(* LS Electric XG5000 project: XMC_CrossCoupled *)
(* project to test Cross Coupled functionality *)
(* PLC LSPLC *)
(* module base 0 slot 0: Input/Output Module:XMC-DN24 (DC 24V Input 8Points/TR output 16Points) *)
(* module base 0 slot 1: Internal Analog Input/Output:XMF-AH04E (A/D voltage/current 2 channels, D/A voltage 2 channels) *)
(* task Periodic Task: Kind=2 *)
(* task Initialization Task: Kind=1 *)
(* task NC Program: Kind=6 *)

PROGRAM Cross_Coupled_ST (* task: Scan Program *)
(* structured text example of cross-coupled control *)
VAR
    Axis1 : UINT := 1; (* variable for axis 1 *)
    Axis2 : UINT := 2; (* axis 2 variable *)
    Connect_ECAT : BOOL; (* command to execute EtherCAT network connection *)
    Disconnect_ECAT : BOOL; (* disconnect the ethercat network *)
    Execute_CrossCoupleOff : BOOL; (* command to turn off cross-coupled control for axis 1 and axis 2 *)
    Execute_CrossCoupleOn : BOOL; (* command to turn on cross-coupling of axis 1 and axis 2 *)
    Execute_Move : BOOL; (* execute move for axis 1 and axis 2 *)
    Execute_MPloopOff : BOOL; (* command to turn off master loop control for axis 1 and 2 *)
    Execute_MPloopOn : BOOL; (* command to execute master control position loop on *)
    INST_Axis1PloopOff : LS_MASTERPLOOPCONTROLOFF; (* fb to turn off master ploop control for axis 1 *)
    INST_Axis1PloopOn : LS_MASTERPLOOPCONTROLON; (* fb for axis 1 master ploop on *)
    INST_Axis1Relative : MC_MOVERELATIVE; (* relative move for axis 1 *)
    INST_Axis2PloopOff : LS_MASTERPLOOPCONTROLOFF; (* fb to turn off master ploop control for axis 2 *)
    INST_Axis2PloopOn : LS_MASTERPLOOPCONTROLON; (* fb for axis 2 master ploop on *)
    INST_Axis2Relative : MC_MOVERELATIVE; (* fb for relative move of axis 2 *)
    INST_Connect : LS_CONNECT; (* ethercat connect FB *)
    INST_CoupleOff : LS_CROSSCOUPLEDCONTROLOFF; (* fb to disable cross-coupling *)
    INST_CoupleOn : LS_CROSSCOUPLEDCONTROLON; (* fb for turning on cross coupling *)
    INST_Disconnect : LS_DISCONNECT; (* fb to disconnect ethercat network *)
    INST_PowerAll : MC_POWERALL; (* fb to power on all axes *)
    Power_On_Axes : BOOL; (* command to power on all axes *)
END_VAR
(* AutomationDirect.com has provided this code for convenience. This sample code is provided "as-is" with no expressed or implied warranty. 
 If the end user includes any of the sample code (in whole or part), it is the user's responsibility to completely modify, integrate, and test any code to ensure it meets all system and 
 safety requirements for the intended application or system. *)

//Function block Calls
INST_Connect(Execute:=Connect_ECAT, ErrorID=>INST_Connect.ErrorID);
INST_Disconnect(Execute:=Disconnect_ECAT, ErrorID=>INST_Disconnect.ErrorID);

INST_PowerAll(Enable:=Power_On_Axes, Status=>INST_PowerAll.Status, Valid=>INST_PowerAll.Valid, ErrorID=>INST_PowerAll.ErrorID);

INST_Axis1PloopOn(Execute:=Execute_MPloopOn, Axis:=Axis1, P_Gain:=1100.0, I_Gain:=600.0, VelFF_Gain:=10000.0, CtrlLimit:=100000000.0, InControl=>INST_Axis1PloopOn.InControl, ErrorID=>INST_Axis1PloopOn.ErrorID);
INST_Axis2PloopOn(Execute:=Execute_MPloopOn, Axis:=Axis2, P_Gain:=1100.0, I_Gain:=600.0, VelFF_Gain:=10000.0, CtrlLimit:=100000000.0, InControl=>INST_Axis2PloopOn.InControl, ErrorID=>INST_Axis2PloopOn.ErrorID);

INST_CoupleOn(Execute:=Execute_CrossCoupleOn, Axis:=Axis1, PairAxis:=Axis2, P_Gain:=1100.0, SlaveMode:=FALSE, InControl=>INST_CoupleOn.InControl, ErrorID=>INST_CoupleOn.ErrorID);

INST_Axis1Relative(Execute:=Execute_Move, Axis:=Axis1, ContinuousUpdate:=FALSE, Distance:=50000.0, Velocity:=500000.0, 
	Acceleration:=500000.0, Deceleration:= 500000.0, Jerk:=10000.0, BufferMode:=0, ErrorID=>INST_Axis1Relative.ErrorID);
	
INST_Axis2Relative(Execute:=Execute_Move, Axis:=Axis2, ContinuousUpdate:=FALSE, Distance:=50000.0, Velocity:=500000.0, 
	Acceleration:=500000.0, Deceleration:= 500000.0, Jerk:=10000.0, BufferMode:=0, ErrorID=>INST_Axis2Relative.ErrorID);
	
INST_Axis1PloopOff(Execute:=Execute_MPloopOff, Axis:=Axis1, ErrorID=>INST_Axis1PloopOff.ErrorID);
INST_Axis2PloopOff(Execute:=Execute_MPloopOff, Axis:=Axis2, ErrorID=>INST_Axis2PloopOff.ErrorID);
INST_CoupleOff(Execute:=Execute_CrossCoupleOff, Axis:=Axis1, PairAxis:=Axis2, ErrorID=>INST_CoupleOff.ErrorID);
END_PROGRAM

PROGRAM Cross_Coupled_LD (* task: Scan Program *)
(* Ladder version of example code. *)
VAR
    Axis1 : UINT := 1; (* variable for axis 1 *)
    Axis2 : UINT := 2; (* axis 2 variable *)
    Connect_ECAT : BOOL; (* command to execute EtherCAT network connection *)
    Disconnect_ECAT : BOOL; (* disconnect the ethercat network *)
    Execute_CrossCoupleOff : BOOL; (* command to turn off cross-coupled control for axis 1 and axis 2 *)
    Execute_CrossCoupleOn : BOOL; (* command to turn on cross-coupling of axis 1 and axis 2 *)
    Execute_Move : BOOL; (* execute move for axis 1 and axis 2 *)
    Execute_MPloopOff : BOOL; (* command to turn off master loop control for axis 1 and 2 *)
    Execute_MPloopOn : BOOL; (* command to execute master control position loop on *)
    INST_Axis1PloopOff : LS_MASTERPLOOPCONTROLOFF; (* fb to turn off master ploop control for axis 1 *)
    INST_Axis1PloopOn : LS_MASTERPLOOPCONTROLON; (* fb for axis 1 master ploop on *)
    INST_Axis1Relative : MC_MOVERELATIVE; (* relative move for axis 1 *)
    INST_Axis2PloopOff : LS_MASTERPLOOPCONTROLOFF; (* fb to turn off master ploop control for axis 2 *)
    INST_Axis2PloopOn : LS_MASTERPLOOPCONTROLON; (* fb for axis 2 master ploop on *)
    INST_Axis2Relative : MC_MOVERELATIVE; (* fb for relative move of axis 2 *)
    INST_Connect : LS_CONNECT; (* ethercat connect FB *)
    INST_CoupleOff : LS_CROSSCOUPLEDCONTROLOFF; (* fb to disable cross-coupling *)
    INST_CoupleOn : LS_CROSSCOUPLEDCONTROLON; (* fb for turning on cross coupling *)
    INST_Disconnect : LS_DISCONNECT; (* fb to disconnect ethercat network *)
    INST_PowerAll : MC_POWERALL; (* fb to power on all axes *)
    Power_On_Axes : BOOL; (* command to power on all axes *)
END_VAR

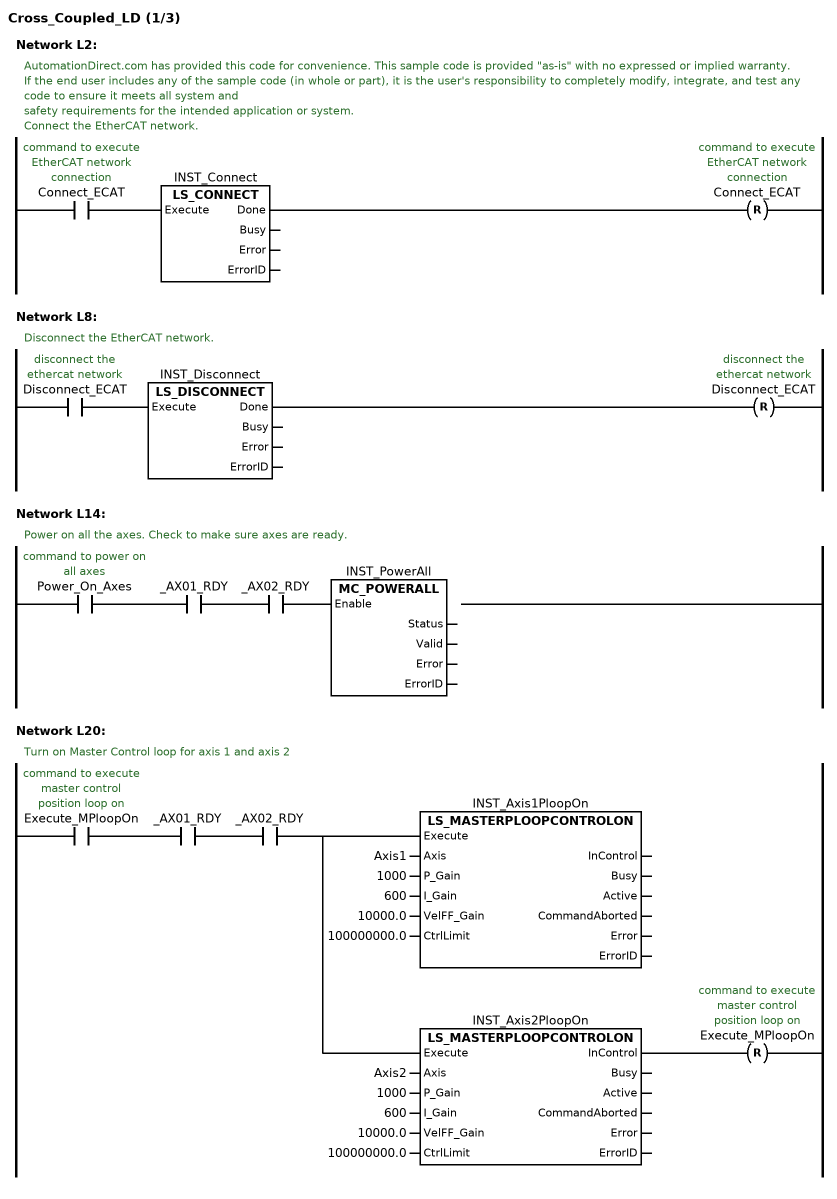
(* AutomationDirect.com has provided this code for convenience. This sample code is provided "as-is" with no expressed or implied warranty. / If the end user includes any of the sample code (in whole or part), it is the user's responsibility to completely modify, integrate, and test any code to ensure it meets all system and / safety requirements for the intended application or system. *)
(* Connect the EtherCAT network. *)
(* Rung L2 *)
INST_Connect(Execute := Connect_ECAT);
IF INST_Connect.Done THEN Connect_ECAT := FALSE; END_IF;
(* Disconnect the EtherCAT network. *)
(* Rung L8 *)
INST_Disconnect(Execute := Disconnect_ECAT);
IF INST_Disconnect.Done THEN Disconnect_ECAT := FALSE; END_IF;
(* Power on all the axes. Check to make sure axes are ready. *)
(* Rung L14 *)
INST_PowerAll(Enable := Power_On_Axes AND _AX01_RDY AND _AX02_RDY);
(* Turn on Master Control loop for axis 1 and axis 2 *)
(* Rung L20 *)
INST_Axis1PloopOn(Execute := Execute_MPloopOn AND _AX01_RDY AND _AX02_RDY, Axis := Axis1, P_Gain := 1000, I_Gain := 600, VelFF_Gain := 10000.0, CtrlLimit := 100000000.0);
INST_Axis2PloopOn(Execute := Execute_MPloopOn AND _AX01_RDY AND _AX02_RDY, Axis := Axis2, P_Gain := 1000, I_Gain := 600, VelFF_Gain := 10000.0, CtrlLimit := 100000000.0);
IF INST_Axis2PloopOn.InControl THEN Execute_MPloopOn := FALSE; END_IF;

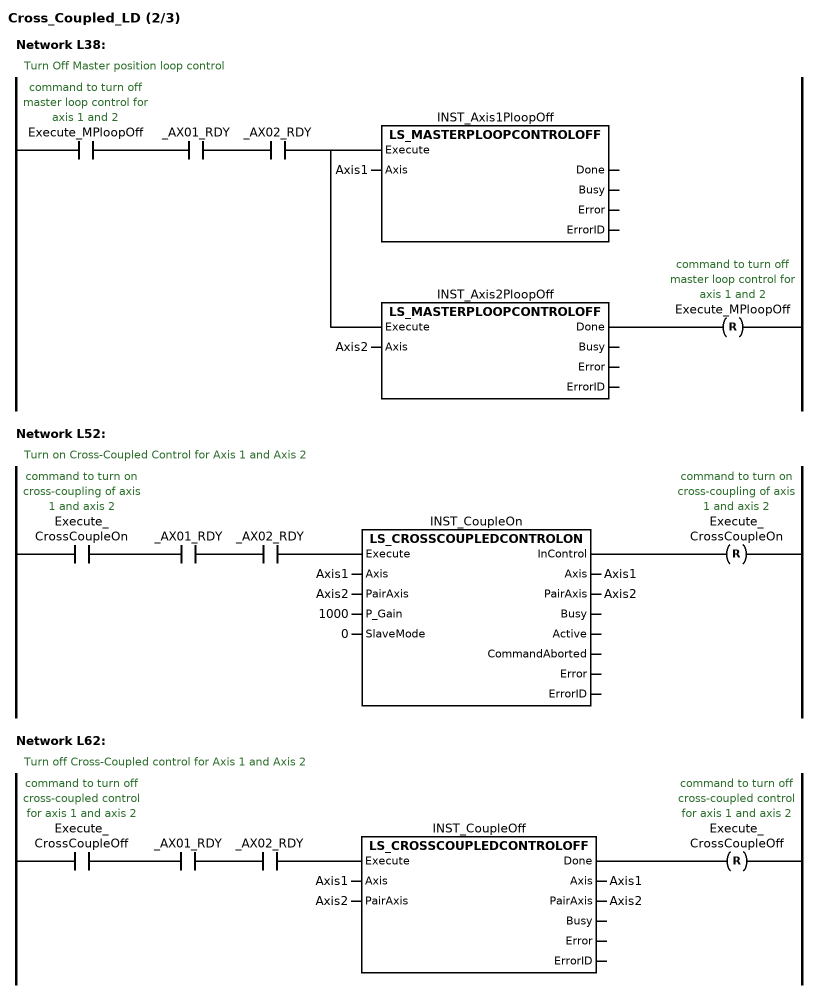
(* Turn Off Master position loop control *)
(* Rung L38 *)
INST_Axis1PloopOff(Execute := Execute_MPloopOff AND _AX01_RDY AND _AX02_RDY, Axis := Axis1);
INST_Axis2PloopOff(Execute := Execute_MPloopOff AND _AX01_RDY AND _AX02_RDY, Axis := Axis2);
IF INST_Axis2PloopOff.Done THEN Execute_MPloopOff := FALSE; END_IF;
(* Turn on Cross-Coupled Control for Axis 1 and Axis 2 *)
(* Rung L52 *)
INST_CoupleOn(Execute := Execute_CrossCoupleOn AND _AX01_RDY AND _AX02_RDY, Axis := Axis1, PairAxis := Axis2, P_Gain := 1000, SlaveMode := 0, Axis => Axis1, PairAxis => Axis2);
IF INST_CoupleOn.InControl THEN Execute_CrossCoupleOn := FALSE; END_IF;
(* Turn off Cross-Coupled control for Axis 1 and Axis 2 *)
(* Rung L62 *)
INST_CoupleOff(Execute := Execute_CrossCoupleOff AND _AX01_RDY AND _AX02_RDY, Axis := Axis1, PairAxis := Axis2, Axis => Axis1, PairAxis => Axis2);
IF INST_CoupleOff.Done THEN Execute_CrossCoupleOff := FALSE; END_IF;

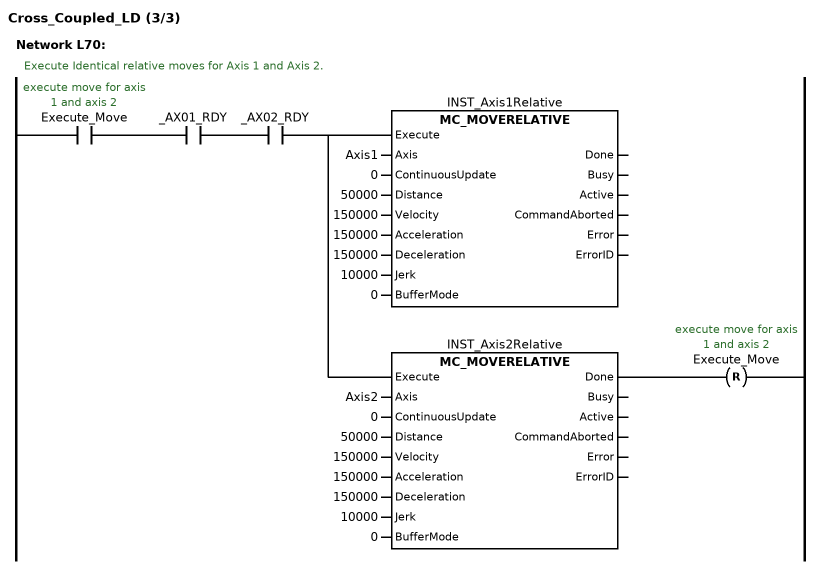
(* Execute Identical relative moves for Axis 1 and Axis 2. *)
(* Rung L70 *)
INST_Axis1Relative(Execute := Execute_Move AND _AX01_RDY AND _AX02_RDY, Axis := Axis1, ContinuousUpdate := 0, Distance := 50000, Velocity := 150000, Acceleration := 150000, Deceleration := 150000, Jerk := 10000, BufferMode := 0);
INST_Axis2Relative(Execute := Execute_Move AND _AX01_RDY AND _AX02_RDY, Axis := Axis2, ContinuousUpdate := 0, Distance := 50000, Velocity := 150000, Acceleration := 150000, Deceleration := 150000, Jerk := 10000, BufferMode := 0);
IF INST_Axis2Relative.Done THEN Execute_Move := FALSE; END_IF;
END_PROGRAM